Yaskawa INFORM job: driller_case_cylinder_program.JBI

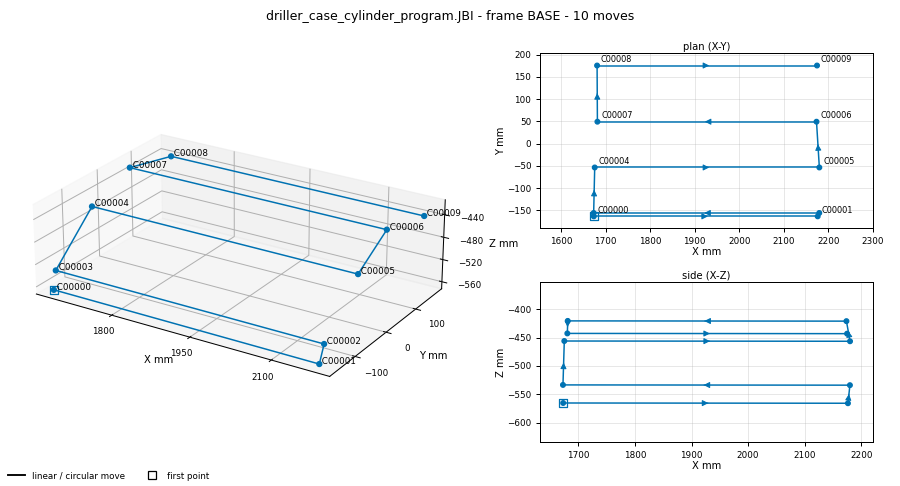
[picture p0: tool path of driller_case_cylinder_program.JBI in frame BASE, 10 of 13 moves have a stored position in this frame; points joined in program order, loops and branches not executed]
/JOB
//NAME driller_case_cylinder_program
//POS
///NPOS 10,0,10,0,0,0
///TOOL 0
///POSTYPE BASE
///RECTAN
///RCONF 0,0,0,0,0,0,0,0,0,0,0,0,0,0,0,0,0,0,0,0,0,0,0,0
C00000=1673.386041,-163.244868,-565.473696,175.000000,-60.000000,90.002202
C00001=2176.206790,-163.244734,-565.924538,175.000000,-60.000000,90.002202
C00002=2179.707290,-155.651275,-534.001856,175.000000,-60.000000,90.023233
C00003=1673.060534,-155.651410,-533.547582,175.000000,-60.000000,90.023233
C00004=1675.421865,-53.453785,-456.041716,-175.000000,-32.366456,90.081071
C00005=2179.906400,-53.453651,-456.494050,-175.000000,-32.366456,90.081071
C00006=2173.550822,49.321224,-420.955530,-174.222357,5.000000,5.000000
C00007=1681.483518,49.321093,-420.514329,-174.222357,5.000000,5.000000
C00008=1680.764354,175.483472,-442.617221,154.347722,5.000000,-5.000000
C00009=2174.696200,175.483603,-443.060093,154.347722,5.000000,-5.000000
///POSTYPE PULSE
///PULSE
EX00000=134144.0
///POSTYPE PULSE
///PULSE
EC00000=134144.0
EC00001=134144.0
EC00002=134144.0
EC00003=134144.0
EC00004=134144.0
EC00005=134144.0
EC00006=134144.0
EC00007=134144.0
EC00008=134144.0
EC00009=134144.0
//INST
///DATE 2023/07/24 11:47
///ATTR SC,RW,RJ
////FRAME BASE
///GROUP1 RB1,ST1
NOP
MOVJ P009 EX000 VJ=15.00
MOVJ C00000 EC00000 VJ=15.0
CALL JOB:SPYON
MOVL C00001 EC00001 V=150.0
MOVL C00002 EC00002 V=150.0
MOVL C00003 EC00003 V=150.0
MOVL C00004 EC00004 V=150.0
MOVL C00005 EC00005 V=150.0
MOVL C00006 EC00006 V=150.0
MOVL C00007 EC00007 V=150.0
MOVL C00008 EC00008 V=150.0
MOVL C00009 EC00009 V=150.0
CALL JOB:SPYOF
MOVJ P009 VJ=15.00
MOVL P009 EX00000 V=150.0
END
